{attribute 'GeneratedUsingTerminal: EK1100-0000-0018'}
{attribute addProperty BoxType "EK1100-0000-0018"}
{attribute addProperty Id "Beckhoff_EL37xxEK1122Beckhoff_EL37xxEK1122_CF4535B32A_0001_EL3702_0000_0002EL3702_8B7B310656A_0002_EL3702_0000_0003EL3702_8B7B310656A_0003_EL3702_0015_0003EL3702_8B7B310656A_0004_EL3742_0000_0001EL3742_09446E4622A_0005_EL3742_0000_0002EL3742_8B7B310656A_0006_EL3742_0000_0003EL3742_8B7B310656A_0007_EL3751_0000_0020EL3751_EB25699D39A_0008_EL3751_0000_0021EL3751_EB25699D39A_0009_EL3751_0000_0022EL3751_EB25699D39A_0010_EL3751_0000_0023EL3751_EB25699D39A_0011_EL3751_0004_0022EL3751_EB25699D39A_0012_EL3751_0004_0023EL3751_EB25699D39A_0013_EL3751_0020_0020EL3751_EB25699D39A_0014_EL3751_0020_0021EL3751_EB25699D39A_0015_EL3751_0020_0022EL3751_EB25699D39A_0016_EL3751_0020_0023EL3751_EB25699D39A_0017_EL3751_0024_0022EL3751_EB25699D39A_0018_EL3751_0024_0023EL3751_EB25699D39A_0019_EL3773_0000_0016EL3773_76254FCD198A_0020_EL3773_0000_0017EL3773_9F446A58198A_0021_EL3773_0000_0018EL3773_B1559BD7192A_0022_EL3773_0000_0019EL3773_89531C23192A_0023_EL3773_0000_0020EL3773_89531C23192A_0024_EL3773_0000_0021EL3773_89531C23192A_0025_EL3783_0000_0018EL3783_BA705D69317"}
{attribute addProperty CRC "2904626126"}
{attribute addProperty Size "2253"}
TYPE Beckhoff_EL37xx_AD2113CE EXTENDS EK1100_AB5A9467 :
STRUCT
	{attribute addProperty Name "Beckhoff_EL37xxEK1122"}
	Beckhoff_EL37xxEK1122 : Beckhoff_EL37xxEK1122_CF4535B3;
	{attribute addProperty Name "A_0001_EL3702_0000_0002"}
	A_0001_EL3702_0000_0002 : EL3702_8B7B3106;
	{attribute addProperty Name "A_0002_EL3702_0000_0003"}
	A_0002_EL3702_0000_0003 : EL3702_8B7B3106;
	{attribute addProperty Name "A_0003_EL3702_0015_0003"}
	A_0003_EL3702_0015_0003 : EL3702_8B7B3106;
	{attribute addProperty Name "A_0004_EL3742_0000_0001"}
	A_0004_EL3742_0000_0001 : EL3742_09446E46;
	{attribute addProperty Name "A_0005_EL3742_0000_0002"}
	A_0005_EL3742_0000_0002 : EL3742_8B7B3106;
	{attribute addProperty Name "A_0006_EL3742_0000_0003"}
	A_0006_EL3742_0000_0003 : EL3742_8B7B3106;
	{attribute addProperty Name "A_0007_EL3751_0000_0020"}
	A_0007_EL3751_0000_0020 : EL3751_EB25699D;
	{attribute addProperty Name "A_0008_EL3751_0000_0021"}
	A_0008_EL3751_0000_0021 : EL3751_EB25699D;
	{attribute addProperty Name "A_0009_EL3751_0000_0022"}
	A_0009_EL3751_0000_0022 : EL3751_EB25699D;
	{attribute addProperty Name "A_0010_EL3751_0000_0023"}
	A_0010_EL3751_0000_0023 : EL3751_EB25699D;
	{attribute addProperty Name "A_0011_EL3751_0004_0022"}
	A_0011_EL3751_0004_0022 : EL3751_EB25699D;
	{attribute addProperty Name "A_0012_EL3751_0004_0023"}
	A_0012_EL3751_0004_0023 : EL3751_EB25699D;
	{attribute addProperty Name "A_0013_EL3751_0020_0020"}
	A_0013_EL3751_0020_0020 : EL3751_EB25699D;
	{attribute addProperty Name "A_0014_EL3751_0020_0021"}
	A_0014_EL3751_0020_0021 : EL3751_EB25699D;
	{attribute addProperty Name "A_0015_EL3751_0020_0022"}
	A_0015_EL3751_0020_0022 : EL3751_EB25699D;
	{attribute addProperty Name "A_0016_EL3751_0020_0023"}
	A_0016_EL3751_0020_0023 : EL3751_EB25699D;
	{attribute addProperty Name "A_0017_EL3751_0024_0022"}
	A_0017_EL3751_0024_0022 : EL3751_EB25699D;
	{attribute addProperty Name "A_0018_EL3751_0024_0023"}
	A_0018_EL3751_0024_0023 : EL3751_EB25699D;
	{attribute addProperty Name "A_0019_EL3773_0000_0016"}
	A_0019_EL3773_0000_0016 : EL3773_76254FCD;
	{attribute addProperty Name "A_0020_EL3773_0000_0017"}
	A_0020_EL3773_0000_0017 : EL3773_9F446A58;
	{attribute addProperty Name "A_0021_EL3773_0000_0018"}
	A_0021_EL3773_0000_0018 : EL3773_B1559BD7;
	{attribute addProperty Name "A_0022_EL3773_0000_0019"}
	A_0022_EL3773_0000_0019 : EL3773_89531C23;
	{attribute addProperty Name "A_0023_EL3773_0000_0020"}
	A_0023_EL3773_0000_0020 : EL3773_89531C23;
	{attribute addProperty Name "A_0024_EL3773_0000_0021"}
	A_0024_EL3773_0000_0021 : EL3773_89531C23;
	{attribute addProperty Name "A_0025_EL3783_0000_0018"}
	A_0025_EL3783_0000_0018 : EL3783_BA705D69;
END_STRUCT
END_TYPE

(* stored: Version 1.2.0.0, ProductVersion 3.1.4024.9
   DUT Beckhoff_EL37xx_AD2113CE: Id {eee6f754-ddeb-459f-8a6b-34138f589c19} *)
